// TIA Portal project "Diagrama_de_Stari" (V15.1)

(* hardware
DEVICE "S71500/ET200MP station_1"  S7-1500 station
   slot 0: "Rail_0"  Rack  6ES7 590-1***0-0AA0
   slot 1: "PLC_1"  CPU 1513-1 PN  6ES7 513-1AL02-0AB0  V2.6
      slot 3: "CPU display_1"  6ES7591-1AA00-0AA0
*)

// ===== PLC "PLC_1"  CPU 1513-1 PN =====

VAR_GLOBAL   // PLC tag table "Default tag table"
   "System_Byte" AT %MB8069 : Byte;
   "FirstScan" AT %M8069.0 : Bool;
   "DiagStatusUpdate" AT %M8069.1 : Bool;
   "AlwaysTRUE" AT %M8069.2 : Bool;
   "AlwaysFALSE" AT %M8069.3 : Bool;
   "Clock_Byte" AT %MB8080 : Byte;
   "Clock_10Hz" AT %M8080.0 : Bool;
   "Clock_5Hz" AT %M8080.1 : Bool;
   "Clock_2.5Hz" AT %M8080.2 : Bool;
   "Clock_2Hz" AT %M8080.3 : Bool;
   "Clock_1.25Hz" AT %M8080.4 : Bool;
   "Clock_1Hz" AT %M8080.5 : Bool;
   "Clock_0.625Hz" AT %M8080.6 : Bool;
   "Clock_0.5Hz" AT %M8080.7 : Bool;
END_VAR

DATA_BLOCK "Variabile"   // DB1
{ S7_Optimized_Access := 'TRUE' }
VERSION : 0.1
   VAR
      stare : Int := 1;
      ETA : Word := 16#0000;
      cmd_shutdown : Bool;
      cmd_switchOn : Bool;
      cmd_switchOn2 : Bool;
      cmd_enableOp : Bool;
      cmd_disableVoltage : Bool;
      cmd_quickStop : Bool;
      cmd_faultReset : Bool;
      sim_fault : Bool;
   END_VAR
BEGIN
END_DATA_BLOCK

// folder: System blocks/Program resources

DATA_BLOCK "timer_franare"   // DB2
{ S7_Optimized_Access := 'TRUE' }
AUTHOR : Simatic
FAMILY : IEC
NAME : IEC_TMR
VERSION : 1.0
// stored: InstanceOfName IEC_TIMER
"IEC_TIMER"
BEGIN
END_DATA_BLOCK

DATA_BLOCK "timere_trecere_s1-s2"   // DB3
{ S7_Optimized_Access := 'TRUE' }
AUTHOR : Simatic
FAMILY : IEC
NAME : IEC_TMR
VERSION : 1.0
// stored: InstanceOfName IEC_TIMER
"IEC_TIMER"
BEGIN
END_DATA_BLOCK

// folder: (top level)

ORGANIZATION_BLOCK "Main"   // OB1, LAD, ProgramCycle
TITLE = "Main Program Sweep (Cycle)"
{ S7_Optimized_Access := 'TRUE' }
VERSION : 0.1
   VAR_INPUT
      Initial_Call : Bool;   // Initial call of this OB
      Remanence : Bool;   // =True, if remanent data are available
   END_VAR
   VAR_TEMP   // added for the SCL form of the ladder/FBD networks
      _w1 : Bool;
   END_VAR
BEGIN

REGION Network 1: daca este in starea 1, not ready to switch on, sa dea automat pe starea 2
   // stare: 1 - not ready to switch on, 2 - disabeled, 3 - ready, 4 - switched on, 5 - operation enabeled, 6 - quick stop, 8 - fault
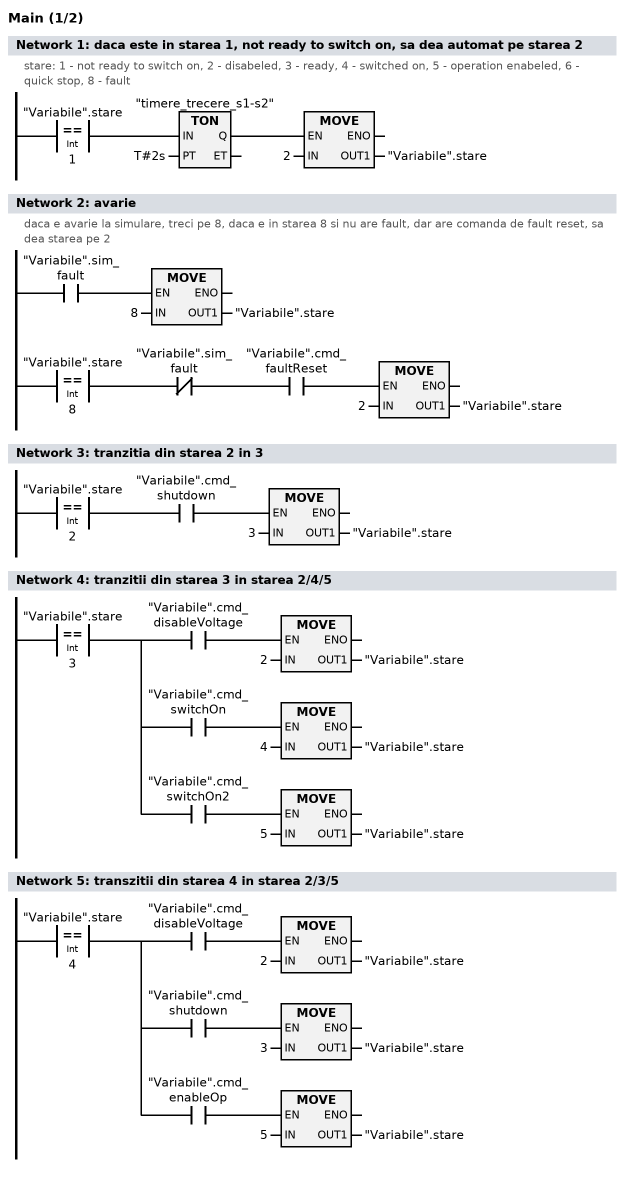
   "timere_trecere_s1-s2".TON(IN := "Variabile".stare = 1, PT := T#2s);
   IF "timere_trecere_s1-s2".Q THEN "Variabile".stare := 2; END_IF;
END_REGION

REGION Network 2: avarie
   // daca e avarie la simulare, treci pe 8, daca e in starea 8 si nu are fault, dar are comanda de fault reset, sa dea starea pe 2
   RUNG wire#powerrail
      Contact( "Variabile".sim_fault )
      Move(in := 8, out1 => "Variabile".stare)
   END_RUNG
   RUNG wire#powerrail
      { S7_Templates := "SrcType := Int" } EQ_Contact(in1 := "Variabile".stare, in2 := 8)
      I_Contact( "Variabile".sim_fault )
      Contact( "Variabile".cmd_faultReset )
      Move(in := 2, out1 => "Variabile".stare)
   END_RUNG
   // the same network as SCL:
   IF "Variabile".sim_fault THEN "Variabile".stare := 8; END_IF;
   IF ("Variabile".stare = 8) AND NOT "Variabile".sim_fault AND "Variabile".cmd_faultReset THEN
       "Variabile".stare := 2;
   END_IF;
END_REGION

REGION Network 3: tranzitia din starea 2 in 3
   RUNG wire#powerrail
      { S7_Templates := "SrcType := Int" } EQ_Contact(in1 := "Variabile".stare, in2 := 2)
      Contact( "Variabile".cmd_shutdown )
      Move(in := 3, out1 => "Variabile".stare)
   END_RUNG
   // the same network as SCL:
   IF ("Variabile".stare = 2) AND "Variabile".cmd_shutdown THEN "Variabile".stare := 3; END_IF;
END_REGION

REGION Network 4: tranzitii din starea 3 in starea 2/4/5
   RUNG wire#powerrail
      { S7_Templates := "SrcType := Int" } EQ_Contact(in1 := "Variabile".stare, in2 := 3)
      wire#w1
      Contact( "Variabile".cmd_disableVoltage )
      Move(in := 2, out1 => "Variabile".stare)
   END_RUNG
   RUNG wire#w1
      Contact( "Variabile".cmd_switchOn )
      Move(in := 4, out1 => "Variabile".stare)
   END_RUNG
   RUNG wire#w1
      Contact( "Variabile".cmd_switchOn2 )
      Move(in := 5, out1 => "Variabile".stare)
   END_RUNG
   // the same network as SCL:
   #_w1 := "Variabile".stare = 3;
   IF #_w1 AND "Variabile".cmd_disableVoltage THEN "Variabile".stare := 2; END_IF;
   IF #_w1 AND "Variabile".cmd_switchOn THEN "Variabile".stare := 4; END_IF;
   IF #_w1 AND "Variabile".cmd_switchOn2 THEN "Variabile".stare := 5; END_IF;
END_REGION

REGION Network 5: transzitii din starea 4 in starea 2/3/5
   RUNG wire#powerrail
      { S7_Templates := "SrcType := Int" } EQ_Contact(in1 := "Variabile".stare, in2 := 4)
      wire#w1
      Contact( "Variabile".cmd_disableVoltage )
      Move(in := 2, out1 => "Variabile".stare)
   END_RUNG
   RUNG wire#w1
      Contact( "Variabile".cmd_shutdown )
      Move(in := 3, out1 => "Variabile".stare)
   END_RUNG
   RUNG wire#w1
      Contact( "Variabile".cmd_enableOp )
      Move(in := 5, out1 => "Variabile".stare)
   END_RUNG
   // the same network as SCL:
   #_w1 := "Variabile".stare = 4;
   IF #_w1 AND "Variabile".cmd_disableVoltage THEN "Variabile".stare := 2; END_IF;
   IF #_w1 AND "Variabile".cmd_shutdown THEN "Variabile".stare := 3; END_IF;
   IF #_w1 AND "Variabile".cmd_enableOp THEN "Variabile".stare := 5; END_IF;
END_REGION

REGION Network 6: tranzitii din starea 5 in starea 2/3/4/6
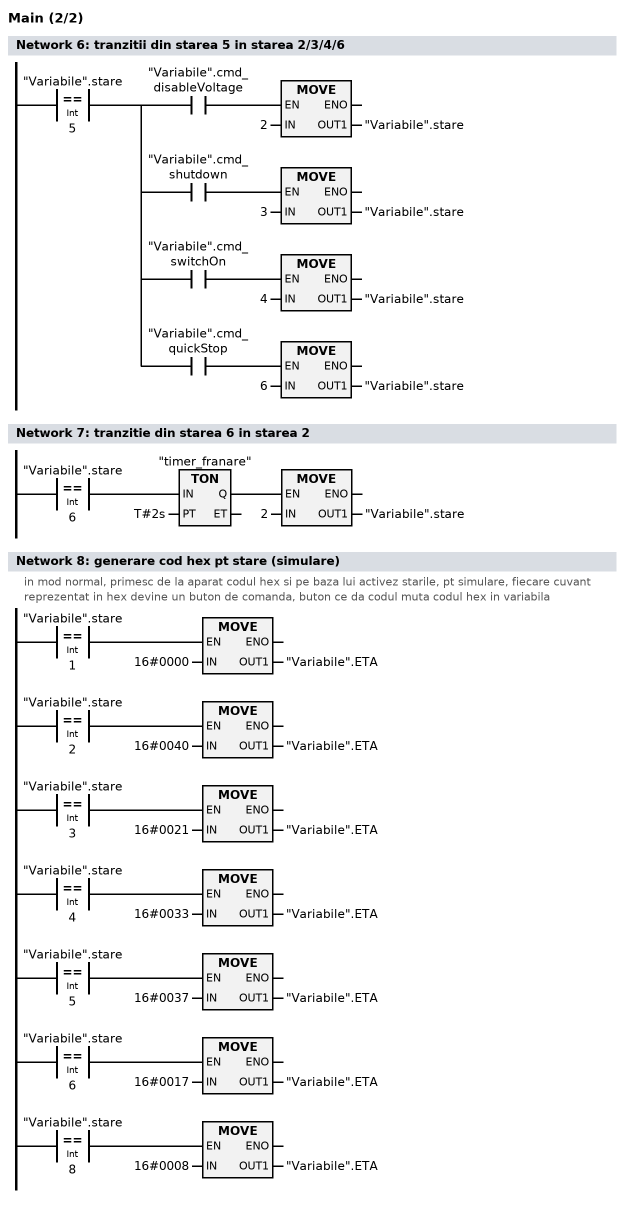
   RUNG wire#powerrail
      { S7_Templates := "SrcType := Int" } EQ_Contact(in1 := "Variabile".stare, in2 := 5)
      wire#w1
      Contact( "Variabile".cmd_disableVoltage )
      Move(in := 2, out1 => "Variabile".stare)
   END_RUNG
   RUNG wire#w1
      Contact( "Variabile".cmd_shutdown )
      Move(in := 3, out1 => "Variabile".stare)
   END_RUNG
   RUNG wire#w1
      Contact( "Variabile".cmd_switchOn )
      Move(in := 4, out1 => "Variabile".stare)
   END_RUNG
   RUNG wire#w1
      Contact( "Variabile".cmd_quickStop )
      Move(in := 6, out1 => "Variabile".stare)
   END_RUNG
   // the same network as SCL:
   #_w1 := "Variabile".stare = 5;
   IF #_w1 AND "Variabile".cmd_disableVoltage THEN "Variabile".stare := 2; END_IF;
   IF #_w1 AND "Variabile".cmd_shutdown THEN "Variabile".stare := 3; END_IF;
   IF #_w1 AND "Variabile".cmd_switchOn THEN "Variabile".stare := 4; END_IF;
   IF #_w1 AND "Variabile".cmd_quickStop THEN "Variabile".stare := 6; END_IF;
END_REGION

REGION Network 7: tranzitie din starea 6 in starea 2
   "timer_franare".TON(IN := "Variabile".stare = 6, PT := T#2s);
   IF "timer_franare".Q THEN "Variabile".stare := 2; END_IF;
END_REGION

REGION Network 8: generare cod hex pt stare (simulare)
   // in mod normal, primesc de la aparat codul hex si pe baza lui activez starile, pt simulare, fiecare cuvant reprezentat in hex devine un buton de comanda, buton ce da codul muta codul hex in variabila
   RUNG wire#powerrail
      { S7_Templates := "SrcType := Int" } EQ_Contact(in1 := "Variabile".stare, in2 := 1)
      Move(in := 16#0000, out1 => "Variabile".ETA)
   END_RUNG
   RUNG wire#powerrail
      { S7_Templates := "SrcType := Int" } EQ_Contact(in1 := "Variabile".stare, in2 := 2)
      Move(in := 16#0040, out1 => "Variabile".ETA)
   END_RUNG
   RUNG wire#powerrail
      { S7_Templates := "SrcType := Int" } EQ_Contact(in1 := "Variabile".stare, in2 := 3)
      Move(in := 16#0021, out1 => "Variabile".ETA)
   END_RUNG
   RUNG wire#powerrail
      { S7_Templates := "SrcType := Int" } EQ_Contact(in1 := "Variabile".stare, in2 := 4)
      Move(in := 16#0033, out1 => "Variabile".ETA)
   END_RUNG
   RUNG wire#powerrail
      { S7_Templates := "SrcType := Int" } EQ_Contact(in1 := "Variabile".stare, in2 := 5)
      Move(in := 16#0037, out1 => "Variabile".ETA)
   END_RUNG
   RUNG wire#powerrail
      { S7_Templates := "SrcType := Int" } EQ_Contact(in1 := "Variabile".stare, in2 := 6)
      Move(in := 16#0017, out1 => "Variabile".ETA)
   END_RUNG
   RUNG wire#powerrail
      { S7_Templates := "SrcType := Int" } EQ_Contact(in1 := "Variabile".stare, in2 := 8)
      Move(in := 16#0008, out1 => "Variabile".ETA)
   END_RUNG
   // the same network as SCL:
   IF "Variabile".stare = 1 THEN "Variabile".ETA := 16#0000; END_IF;
   IF "Variabile".stare = 2 THEN "Variabile".ETA := 16#0040; END_IF;
   IF "Variabile".stare = 3 THEN "Variabile".ETA := 16#0021; END_IF;
   IF "Variabile".stare = 4 THEN "Variabile".ETA := 16#0033; END_IF;
   IF "Variabile".stare = 5 THEN "Variabile".ETA := 16#0037; END_IF;
   IF "Variabile".stare = 6 THEN "Variabile".ETA := 16#0017; END_IF;
   IF "Variabile".stare = 8 THEN "Variabile".ETA := 16#0008; END_IF;
END_REGION
END_ORGANIZATION_BLOCK